{attribute 'qualified_only'}
VAR_GLOBAL CONSTANT
	ERROR_IF_NC_AXIS_IS_NOT_MAPPED : BOOL := TRUE;
END_VAR

(* stored: Version 1.1.0.1, ProductVersion 3.1.4024.12
   GVL NcParameterlist: Id {7d7982ad-c533-4f25-8308-395a4bad6e48}, ParameterList True *)
